CASE nState OF
    // Start by setting everything to a known value
    INIT:
        nState := WAIT_EXEC;
        bError := FALSE;
        sErrorMessage := '';
        bDone := FALSE;
        bCausedError := FALSE;
    // Normal "waiting for move command" state
    WAIT_EXEC:
        bMyMove := FALSE;
        // Looking for a rising edge on bExecute
        IF rtExec.Q THEN
            bDone := FALSE;
            nState := PICK_REQUEST;
        END_IF
    // Decide how to handle the request
    PICK_REQUEST:
        IF stMotionStage.bBusy THEN
            CASE enumMotionRequest OF
                ENUM_MotionRequest.WAIT:
                    nState := WAIT_OTHER_MOVE;
                ENUM_MotionRequest.INTERRUPT:
                    nState := STOP_OTHER_MOVE;
                ENUM_MotionRequest.ABORT:
                    nState := ERROR;
                    bError := TRUE;
                    nErrorId := 16#7900;
            END_CASE
        ELSE
            nState := START_MOVE;
        END_IF
    // Watch the other move, then see if it's our turn
    WAIT_OTHER_MOVE:
        IF NOT stMotionStage.bBusy THEN
            // Try to pick request again next cycle once the move is over
            nState := PICK_REQUEST;
        END_IF
    // Interrupt the other move, then go to start ours
    STOP_OTHER_MOVE:
        stMotionStage.bExecute := FALSE;
        IF NOT stMotionStage.bBusy THEN
            nState := START_MOVE;
        END_IF
    // Set the correct values on DUT_MotionStage to start a new absolute move
    START_MOVE:
        bMyMove := TRUE;
        stMotionStage.bExecute := TRUE;
        stMotionStage.nCommand := ENUM_EpicsMotorCmd.MOVE_ABSOLUTE;
        stMotionStage.fPosition := fPos;
        stMotionStage.fVelocity := fVel;
        stMotionStage.fAcceleration := fAcc;
        stMotionStage.fDeceleration := fDec;
        nState := WAIT_MY_MOVE;
    // Watch our ongoing move, look for the move to end or requests to stop the move from this FB
    WAIT_MY_MOVE:
        ftBusy(CLK:=stMotionStage.bBusy);
        IF ftBusy.Q THEN
            nState := DONE_MOVING;
        END_IF
        // Implement stop on falling trigger
        IF ftExec.Q THEN
            nState := STOP_MY_MOVE;
        END_IF
    // Request a stop and wait for it to happen
    STOP_MY_MOVE:
        stMotionStage.bExecute := FALSE;
        IF NOT stMotionStage.bBusy THEN
            nState := DONE_MOVING;
        END_IF
    // Pick out the bDone state and return to waiting
    DONE_MOVING:
        bDone := stMotionStage.bDone;
        nState := WAIT_EXEC;
    // Lock us into the error state until the FB is reset
    ERROR:
        bMyMove := FALSE;
END_CASE

// Transition to the ERROR state if applicable
IF bMyMove AND stMotionStage.bError THEN
    nState := ERROR;
    bError := TRUE;
    nErrorId := stMotionStage.nErrorId;
    bCausedError := TRUE;
END_IF
sErrorMessage := F_MotionErrorCodeLookup(nErrorId := nErrorId);

CASE nState OF
INIT, WAIT_EXEC, ERROR:
    bBusy := FALSE;
ELSE
    bBusy := TRUE;
END_CASE

END_FUNCTION_BLOCK

// POUs/Motion/States/FB_PositionStateLock
FUNCTION_BLOCK FB_PositionStateLock
(*
    Implements immutability for a locked DUT_PositionState
    Once this is called the first time, the parameters at the time of the call will be restored on all subsequent calls.
*)
VAR_IN_OUT
    stPositionState: DUT_PositionState;
END_VAR
VAR
    stCachedPositionState: DUT_PositionState;
    bInit: BOOL := FALSE;
END_VAR

// Force values to be cached if we've cached something
IF bInit AND stPositionState.bLocked THEN
    stPositionState.sName := stCachedPositionState.sName;
    stPositionState.fPosition := stCachedPositionState.fPosition;
    stPositionState.fDelta := stCachedPositionState.fDelta;
    stPositionState.fVelocity := stCachedPositionState.fVelocity;
    stPositionState.fAccel := stCachedPositionState.fAccel;
    stPositionState.fDecel := stCachedPositionState.fDecel;
// If we haven't cached and we should, make the cache. Note that we skip bLocked, bValid, and bMoveOk
ELSIF NOT bInit AND stPositionState.bLocked THEN
    stCachedPositionState.sName := stPositionState.sName;
    stCachedPositionState.fPosition := stPositionState.fPosition;
    stCachedPositionState.fDelta := stPositionState.fDelta;
    stCachedPositionState.fVelocity := stPositionState.fVelocity;
    stCachedPositionState.fAccel := stPositionState.fAccel;
    stCachedPositionState.fDecel := stPositionState.fDecel;
    bInit := TRUE;
// Do nothing, or unlock the state if bLocked goes FALSE
ELSIF NOT stPositionState.bLocked THEN
    bInit := FALSE;
END_IF

END_FUNCTION_BLOCK

// POUs/Motion/FB_MotionPneumaticActuator
(*This function blcok implements a pnuematic actuator. That can be signle or double acting by setting the ibSingleCntrl accordingly*)
(* with double acting ibCntrlHold signal should be false, while with single acting the signal should be true*)
FUNCTION_BLOCK FB_MotionPneumaticActuator
VAR_INPUT
    (*EPS Interlock Bits*)
    ibInsertOK: BOOL; (*Actuator can be Inserted*)
    ibRetractOK: BOOL; (*ACtuator can be retracted*)
    ibPMPS_OK:BOOL; (*to be linked the Arbiter bit*)
    ibSingleCntrl:BOOL;(* TRUE if Actuator requires one Output signal to be activated, FALSE if its double acting i.e two outputs are required*)
    ibCntrlHold:BOOL; (* Control Signal must retain its value, must be TRUE in the case of single acting*)
    ibOverrideInterlock:BOOL; (*if true interlocks are ignored*)
    // Reset fault
    {attribute 'pytmc' := '
    pv: FF_Reset
    '}
    i_xReset: BOOL;
END_VAR
VAR_OUTPUT
    {attribute 'pytmc' := '
    pv:
    '}
    stPneumaticActuator    :    DUT_MotionPneumaticActuator;
    {attribute 'pytmc' := '
     pv: MPS_OK
     field: ZNAM FALSE
     field: ONAM TRUE
     field: DESC TRUE if MPS signal is OK
    '}
    xMPS_OK:BOOL;
END_VAR
VAR_IN_OUT
    io_fbFFHWO    :    FB_HardwareFFOutput;
END_VAR
VAR
    // PMPS
    fbFF    :    FB_FastFault :=(
        i_DevName := 'MPA',
        i_Desc := 'Fault occurs when the device is moving',
        i_TypeCode := 10#1010);

    (*Init*)
    xFirstPass    :    BOOL;
    fbFSInit        :    R_TRIG;

    (* Timeouts*)
    tTimeOutDuration: TIME:= T#10S;
    tInserttimeout: TON;
    tRetracttimeout:TON;
    (*Limit switch latch timer*)
    tLimitSwitchLatchDuration: TIME:=T#1S;
    tInsertLimitSwitch:TON;
    tRetractLimitSwitch:TON;

    (*Logging*)
    fbLogger : FB_LogMessage := (eSubsystem:=E_SubSystem.MOTION);
    ePrevState : ENUM_PnuematicActuatorPositionState;
    tAction : R_TRIG; // Primary action of this device (Insert_DO, Retract_DO, etc.)
    tOverrideActivated : R_TRIG;

    (*IO*)
    i_xInsertedLS    AT%I*: BOOL;
    i_xRetractedLS    AT%I*: BOOL;
    q_xInsert_DO    AT%Q*: BOOL;
    q_xRetract_DO    AT%Q*: BOOL;

END_VAR


(*Initialize*)
fbFSInit( CLK := TRUE, Q => xFirstPass);
IF xFirstPass THEN
    stPneumaticActuator.eState := ENUM_PnuematicActuatorPositionState.INVALID;
    stPneumaticActuator.bRetract_SW := FALSE;
    stPneumaticActuator.bInsert_SW := FALSE;
END_IF

(*Soft IO Mapping to EPICS PVs*)
ACT_IO();

(* Manage States*)
IF stPneumaticActuator.i_bInLimitSwitch AND  stPneumaticActuator.i_bOutLimitSwitch THEN
    stPneumaticActuator.eState:=ENUM_PnuematicActuatorPositionState.INVALID;
ELSIF NOT stPneumaticActuator.i_bInLimitSwitch AND stPneumaticActuator.i_bOutLimitSwitch THEN
    stPneumaticActuator.eState:=ENUM_PnuematicActuatorPositionState.RETRACTED;
ELSIF stPneumaticActuator.i_bInLimitSwitch AND NOT stPneumaticActuator.i_bOutLimitSwitch THEN
    stPneumaticActuator.eState:=ENUM_PnuematicActuatorPositionState.INSERTED;
ELSIF NOT stPneumaticActuator.i_bInLimitSwitch AND NOT stPneumaticActuator.i_bOutLimitSwitch THEN
    stPneumaticActuator.eState:=ENUM_PnuematicActuatorPositionState.MOVING;
ELSE
    stPneumaticActuator.eState:=ENUM_PnuematicActuatorPositionState.INVALID ;
END_IF

(*Set the Done/Busy signal*)
stPneumaticActuator.bDone := (stPneumaticActuator.bRetract_SW AND stPneumaticActuator.eState=ENUM_PnuematicActuatorPositionState.RETRACTED)
                            OR (stPneumaticActuator.bInsert_SW AND stPneumaticActuator.eState=ENUM_PnuematicActuatorPositionState.INSERTED);
stPneumaticActuator.bBusy := (stPneumaticActuator.bRetract_SW AND stPneumaticActuator.eState<>ENUM_PnuematicActuatorPositionState.RETRACTED)
                            OR (stPneumaticActuator.bInsert_SW AND stPneumaticActuator.eState<>ENUM_PnuematicActuatorPositionState.INSERTED);
(*MPS FAULT*)
(* MPS Faults when the actuator is in motion*)
xMPS_OK := (stPneumaticActuator.eState=ENUM_PnuematicActuatorPositionState.RETRACTED) OR (stPneumaticActuator.eState=ENUM_PnuematicActuatorPositionState.INSERTED);
(*PMPS PERMISSION*)
// yet to be implemented

(* Can't have bRetract_SW and  bInsert_SW both be true*)
If (stPneumaticActuator.bRetract_SW) AND (stPneumaticActuator.bInsert_SW) THEN
    stPneumaticActuator.bRetract_SW := FALSE;
    stPneumaticActuator.bInsert_SW := FALSE;
END_IF
//Redundant??
(*Check if both digital outputs active at the same time, and clear all*)
IF stPneumaticActuator.q_bInsert THEN
    stPneumaticActuator.q_bRetract := FALSE;
    stPneumaticActuator.bRetract_SW:= FALSE;
END_IF;
IF stPneumaticActuator.q_bRetract THEN
    stPneumaticActuator.q_bInsert := FALSE;
    stPneumaticActuator.bInsert_SW:= FALSE;
END_IF;

(*Actuate the device*)
stPneumaticActuator.q_bRetract := stPneumaticActuator.bRetractOK AND stPneumaticActuator.bRetract_SW AND NOT stPneumaticActuator.bInsert_SW ;
stPneumaticActuator.q_bInsert := stPneumaticActuator.bInsertOK AND stPneumaticActuator.bInsert_SW AND NOT stPneumaticActuator.bRetract_SW ;

(*Reset the Control signal when command has been executed and give time to ensure the actuator is fully seated in either direction*)
IF (NOT ibSingleCntrl AND NOT ibCntrlHold) THEN
   IF (stPneumaticActuator.bRetract_SW AND stPneumaticActuator.i_bOutLimitSwitch AND tRetractLimitSwitch.Q ) THEN stPneumaticActuator.q_bRetract := FALSE; END_IF
   IF (stPneumaticActuator.bInsert_SW AND stPneumaticActuator.i_bInLimitSwitch AND tInsertLimitSwitch.Q) THEN stPneumaticActuator.q_bInsert := FALSE; END_IF
END_IF

(*Timers*)
tInserttimeout(IN:= stPneumaticActuator.q_bInsert, PT := tTimeOutDuration );
tRetracttimeout(IN:= stPneumaticActuator.q_bRetract, PT := tTimeOutDuration);
tInsertLimitSwitch(IN:= stPneumaticActuator.i_bInLimitSwitch, PT := tLimitSwitchLatchDuration);
tRetractLimitSwitch(IN:= stPneumaticActuator.i_bOutLimitSwitch, PT := tLimitSwitchLatchDuration);


///Check moving postion timout
IF NOT stPneumaticActuator.i_bInLimitSwitch AND tInserttimeout.Q THEN
    stPneumaticActuator.bError := TRUE;
    stPneumaticActuator.sErrorMessage:= 'Actuator insert timeout';
ELSIF NOT stPneumaticActuator.i_bOutLimitSwitch AND tRetracttimeout.Q THEN
    stPneumaticActuator.bError := TRUE;
    stPneumaticActuator.sErrorMessage:= 'Actuator retract timeout';
END_IF
// Reset error
stPneumaticActuator.bError R= stPneumaticActuator.bReset;

(*FAST FAULT*)
fbFF(i_xOK := xMPS_OK,
    i_xReset := i_xReset,
    io_fbFFHWO := io_fbFFHWO);

(*Soft IO Mapping to Epics pvs*)
ACT_IO();

ACTION ACT_IO:
(*Inputs*)
stPneumaticActuator.i_bInLimitSwitch :=  i_xInsertedLS;
stPneumaticActuator.i_bOutLimitSwitch := i_xRetractedLS;

(*outputs*)
q_xInsert_DO:=stPneumaticActuator.q_bInsert;
q_xRetract_DO:=stPneumaticActuator.q_bRetract;

(*EPICS*)
stPneumaticActuator.bRetractOK := ibRetractOK;
stPneumaticActuator.bInsertOK := ibInsertOK;
END_ACTION

ACTION ACT_Logger:
// Log Valve timeouts
IF (tInserttimeout.Q OR tRetracttimeout.Q) THEN fbLogger(sMsg:=stPneumaticActuator.sErrorMessage, eSevr:=TcEventSeverity.Warning); END_IF

// Log Actuator commands
// Log valve open
tAction(CLK:= (stPneumaticActuator.q_bRetract OR stPneumaticActuator.q_bInsert));
IF tAction.Q THEN
   IF(stPneumaticActuator.q_bRetract) THEN fbLogger(sMsg:='Actuator commanded retract', eSevr:=TcEventSeverity.Info); END_IF
   IF(stPneumaticActuator.q_bInsert) THEN fbLogger(sMsg:='Actuator commanded insert', eSevr:=TcEventSeverity.Info); END_IF
END_IF


// State Logging
IF ePrevState <> stPneumaticActuator.eState THEN
      CASE stPneumaticActuator.eState OF
        ENUM_PnuematicActuatorPositionState.INVALID:
            fbLogger(sMsg:='Actuator invalid position.', eSevr:=TcEventSeverity.Critical);
          ENUM_PnuematicActuatorPositionState.MOVING:
            fbLogger(sMsg:='Actuator moving', eSevr:=TcEventSeverity.Warning);
        ENUM_PnuematicActuatorPositionState.RETRACTED:
            fbLogger(sMsg:='Actuator Retracted.', eSevr:=TcEventSeverity.Info);
        ENUM_PnuematicActuatorPositionState.INSERTED:
            fbLogger(sMsg:='Actuator Inserted.', eSevr:=TcEventSeverity.Info);
      END_CASE
      ePrevState := stPneumaticActuator.eState;
  END_IF
END_ACTION

END_FUNCTION_BLOCK

// POUs/Motion/FB_MotionStageSim
FUNCTION_BLOCK FB_MotionStageSim
(*
    Set all the values needed for a fake motor to be movable
    via the IOC, then call FB_MotionStage
*)
VAR_IN_OUT
    stMotionStage: DUT_MotionStage;
END_VAR
VAR
    fbMotionStage: FB_MotionStage;
    bInit: BOOL;
END_VAR

IF NOT bInit THEN
    bInit := TRUE;
    // Stand-in for no forward limit
    stMotionStage.bLimitForwardEnable := TRUE;
    // Stand-in for no reverse limit
    stMotionStage.bLimitBackwardEnable := TRUE;
    // Stand-in for no STO button
    stMotionStage.bHardwareEnable := TRUE;
    // Stand-in for no PMPS governer
    stMotionStage.bPowerSelf := TRUE;
    // Always keep it enabled for testing ease
    stMotionStage.nEnableMode := ENUM_StageEnableMode.ALWAYS;
END_IF
// Call FB_MotionStage to do the thing
fbMotionStage(stMotionStage := stMotionStage);

END_FUNCTION_BLOCK

// POUs/MotorTesting/FB_MicroStepCountTest
FUNCTION_BLOCK FB_MicroStepCountTest
VAR_INPUT
    bExecute: BOOL;
    fStepSize: LREAL;
    nSteps: UINT;
    fMicroStep: LREAL;
    fVelocity: LREAL;
    tSettleTime: TIME;
END_VAR
VAR_IN_OUT
    Axis: AXIS_REF;
END_VAR
VAR_OUTPUT
    nStepsCounted: UINT;
    nTheorySteps: UINT;
    fPercent: LREAL;
    fEstMicroSize: LREAL;
END_VAR
VAR
    fbMoveRel: MC_MoveRelative;
    fbSettleTimer: TON;
    bDoMove: BOOL;
    nStepCounter: UINT;

    arrPosBuffer: ARRAY [0..99] OF LREAL;
    fAvgPos: LREAL;
    nArrIndex: UINT;
    nLoopIndex: UINT;

    fStartPos: LREAL;
    fPrevPos: LREAL;
    fStepChange: LREAL;

    fStepSum: LREAL;
END_VAR

// Motion FB
fbMoveRel(Axis:=Axis,
    Execute:=bDoMove,
    Distance:=fStepSize,
    Velocity:=fVelocity);

// Settle time
fbSettleTimer(IN:=fbMoveRel.Done,
    PT:=tSettleTime);

// Re-enable the move for next cycle
bDoMove := bExecute AND nStepCounter < nSteps;

// Calculate rolling average
arrPosBuffer[nArrIndex] := Axis.NcToPlc.ActPos;
fAvgPos := 0;
FOR nLoopIndex := 0 TO 99 DO
    fAvgPos := fAvgPos + arrPosBuffer[nLoopIndex];
END_FOR;
fAvgPos := fAvgPos / 100;
nArrIndex := (nArrIndex + 1) MOD 100;

// Initialize starting variables
IF NOT bExecute THEN
    fStartPos := fAvgPos;
    fPrevPos := fAvgPos;
END_IF

// Check results
IF fbSettleTimer.Q THEN
    fStepChange := fAvgPos - fPrevPos;
    // Invert fStepChange if we were doing negative steps
    IF fStepSize < 0 THEN
        fStepChange := fStepChange * -1;
    END_IF
    IF fStepChange > fMicroStep * 0.5 THEN
        nStepsCounted := nStepsCounted + 1;
        fStepSum := fStepSum + fStepChange;
        fEstMicroSize := fStepSum / nStepsCounted;
    END_IF
    nTheorySteps := DINT_TO_UINT(TRUNC(ABS((fStartPos - fAvgPos) / fMicroStep)));
    IF nTheorySteps > 0 THEN
        fPercent := 100 * nStepsCounted / nTheorySteps;
    END_IF
    fPrevPos := fAvgPos;
    nStepCounter := nStepCounter + 1;
    // Reset the move block
    bDoMove := FALSE;
END_IF

END_FUNCTION_BLOCK

// tc_mca_std_lib/POUs/ErrorHandling/FB_ErrorList
FUNCTION_BLOCK FB_ErrorList

VAR_INPUT
	En : BOOL;											//Enable input
	bReset : BOOL;										//Delete all Error entry
	lErrorID : ULINT;									//ErrorID to be acknoledged
	bACK : BOOL;										//Acknoledge the given error and delete it from the list
END_VAR
	
VAR_OUTPUT
	EnO : BOOL;											//Enable output
	nNoError: UINT;										//Number of Errors
	nNoOverflow : INT;									//Number of Overflows
	pErrorSystem : POINTER TO ST_ErrorSystem;			//Pointer to ErrorSystem
END_VAR

VAR
	nFreePos : UINT;									//Number of free position in the list
	nListCnt1 : UINT;									//work variable
	ErrorSystem : ST_ErrorSystem;						//Data structure of the Error list
END_VAR

(*
* ================================================================================
*                                   DESCRIPTION
* ================================================================================
* This Function Block implements the core structure of the Error/Warning Handling
* system. It realizes the datastructure containing every Error Entry, collect
* statistics about the usage and manage the Error Entries.
* Note: The system is under development, most of the functionalities are not
* implemented or existing functionalities may change with time.
* ================================================================================
*)
EnO := En;

//Ponter to ErrorSystem
pErrorSystem := ADR(ErrorSystem);

//Number of overflows
nNoOverflow := ErrorSystem.nNoOverflows;

IF bReset THEN
	MEMSET ( ADR(ErrorSystem.aErrorData[0]), 0, GVL_ErrorSystem.cSizeOfErrorData * SIZEOF(DUT_TerminalError));
	ErrorSystem.lNextErrorID := 1;
END_IF

//Number of errors in the system
nNoError := 0;
FOR nListCnt1 := 0 TO GVL_ErrorSystem.cSizeOfErrorData - 1 DO
	IF ErrorSystem.aErrorData[nListCnt1].Error_ID <> 0  THEN
		nNoError := nNoError+1; 
	END_IF
END_FOR
ErrorSystem.nNoErrors := nNoError;

//Number of free position in the list
nFreePos := GVL_ErrorSystem.cSizeOfErrorData - nNoError;

//Acknoledge specified Error entry
IF bACK THEN
	FOR nListCnt1 := 0 TO GVL_ErrorSystem.cSizeOfErrorData - 1 DO
		IF ErrorSystem.aErrorData[nListCnt1].Error_ID = lErrorID THEN
			ErrorSystem.aErrorData[nListCnt1].ErrorState := DUT_ErrorState.Acknowledged;
		END_IF
	END_FOR
END_IF

//Deleting acknoledged errors
FOR nListCnt1 := 0 TO GVL_ErrorSystem.cSizeOfErrorData - 1 DO
	IF ErrorSystem.aErrorData[nListCnt1].ErrorState = DUT_ErrorState.Acknowledged THEN
		MEMMOVE (ADR(ErrorSystem.aErrorData[nListCnt1]), ADR(ErrorSystem.aErrorData[nListCnt1+1]), (GVL_ErrorSystem.cSizeOfErrorData - 1 - nListCnt1) * SIZEOF(DUT_TerminalError));
		MEMSET(ADR(ErrorSystem.aErrorData[GVL_ErrorSystem.cSizeOfErrorData - 1]), 0, SIZEOF(DUT_TerminalError));
	END_IF
END_FOR

END_FUNCTION_BLOCK

// tc_mca_std_lib/POUs/ErrorHandling/FB_TerminalError
FUNCTION_BLOCK FB_TerminalError

VAR_INPUT
	En					: BOOL;
	iTerminal_ID		: INT;
	bWcState			: BOOL;
	uiInfoData_State	: UINT;
	pErrorSystem		: POINTER TO ST_ErrorSystem;					//Pointer to the error system
END_VAR

VAR_OUTPUT
	EnO : BOOL;
	bError : BOOL := FALSE;
END_VAR

VAR
	iStateError : UINT;
	iOtherError : UINT;
	ErrorData	: DUT_TerminalError;
	nErrSysCNT	: UINT;
	
	//testing
	bStateChanged : BOOL;						//Indicate if state change happened
	uiInfoData_State_Prev : UINT := 16#8;		//Previous value of Infodata.State
	bWcState_Prev : BOOL := FALSE;				//Previous state of WcState
	
	//FB-s
	
END_VAR

(*
Currently:

Problem:

TODO:

*)

//Connect EN to EnO
EnO:=En;

//Check if pointer is OK
IF pErrorSystem=0 THEN RETURN; END_IF

//Any difference from normal state creates an error
IF En AND (bWcState OR uiInfoData_State<>16#8) THEN
	bError:=TRUE;
ELSE
	bError:=FALSE;
END_IF

//Change detection
IF uiInfoData_State <> uiInfoData_State_Prev OR bWcState <> bWcState_Prev THEN
	bStateChanged := TRUE;
ELSE
	bStateChanged := FALSE;
END_IF

//Update previous values
uiInfoData_State_Prev := uiInfoData_State;
bWcState_Prev := bWcState;

//Decision tree
IF bStateChanged THEN
	IF bError THEN
		IF ErrorData.ErrorState = DUT_ErrorState.Active THEN
			//Close active error
			//Read system time
			ErrorData.nDateTimeOff := Tc2_EtherCAT.F_GetActualDcTime64();
			ErrorData.sDateTimeOff := Tc2_EtherCat.DCTIME64_TO_STRING(ErrorData.nDateTimeOff);
			ErrorData.ErrorState := DUT_ErrorState.Inactive;
			//Write Off-time to Error System
			FOR nErrSysCNT := 0 TO GVL_ErrorSystem.cSizeOfErrorData - 1 DO
				IF pErrorSystem^.aErrorData[nErrSysCNT].Error_ID = ErrorData.Error_ID THEN
					pErrorSystem^.aErrorData[nErrSysCNT].nDateTimeOff := ErrorData.nDateTimeOff;
					pErrorSystem^.aErrorData[nErrSysCNT].sDateTimeOff := ErrorData.sDateTimeOff;
					pErrorSystem^.aErrorData[nErrSysCNT].ErrorState := DUT_ErrorState.Inactive;
					EXIT;
				END_IF
			END_FOR
				
			//Clear ErrorData
			MEMSET(ADR(ErrorData), 0, SIZEOF(ErrorData));
		END_IF
		
		//Open a new error
		ErrorData.ErrorState := DUT_ErrorState.Active;												//Set Error State
		ErrorData.nDateTimeOn := Tc2_EtherCAT.F_GetActualDcTime64();								//Get system time
		ErrorData.sDateTimeOn := Tc2_EtherCat.DCTIME64_TO_STRING(ErrorData.nDateTimeOn);			//Convert to string
		ErrorData.iTerminalID := iTerminal_ID;														//Terminal_ID
		ErrorData.bWcState := bWcState;																//WcState bit
		ErrorData.uiInfoDataState := uiInfoData_State;												//uiInfoData_State
		
		//Error message according to uiInfoData_State and WcState
		iStateError := (uiInfoData_State AND 16#000F);												//Mask for operation state 
		iOtherError := (uiInfoData_State AND 16#00F0);												//Mask for the other 3 kind of errors
		//Error messages according to the least significant digit
		CASE iStateError OF
			16#0001 : ErrorData.sErrorMessage := 'Slave in INIT state;   ';
			16#0002 : ErrorData.sErrorMessage := 'Slave in PREOP state;   ';
			16#0003 : ErrorData.sErrorMessage := 'Slave in BOOT state;   ';
			16#0004 : ErrorData.sErrorMessage := 'Slave in SAFEOP state;   ';
			16#0008 : ;																			//Normal operation state
		ELSE
			ErrorData.sErrorMessage := 'Undefined State of operation;   ';						//I hope we will never see this message
			ErrorData.sErrorMessage := CONCAT (ErrorData.sErrorMessage, UINT_TO_STRING(iStateError));
			ErrorData.sErrorMessage := CONCAT (ErrorData.sErrorMessage, '   ');
		END_CASE
		
		//Error messages according to the second least significant digit
		CASE iOtherError OF
			16#0000 : ;																			//No error case
			16#0010 : ErrorData.sErrorMessage := CONCAT (ErrorData.sErrorMessage, 'Slave signals error;   ');
			16#0020 : ErrorData.sErrorMessage := CONCAT (ErrorData.sErrorMessage, 'Invalid vendorID/productCode read;   ');
			16#0040 : ErrorData.sErrorMessage := CONCAT (ErrorData.sErrorMessage, 'Initialisation error occured;   ');
		ELSE
			ErrorData.sErrorMessage := CONCAT (ErrorData.sErrorMessage, 'Undefined Error ID: ');
			ErrorData.sErrorMessage := CONCAT (ErrorData.sErrorMessage, UINT_TO_STRING(iOtherError));
			ErrorData.sErrorMessage := CONCAT (ErrorData.sErrorMessage, '   ');
		END_CASE
	
		//Errormessage according to WcState bit
		IF bWcState THEN
			ErrorData.sErrorMessage := CONCAT (ErrorData.sErrorMessage, 'Invalid Data;');
		END_IF
		
		//Check for overflow
		IF pErrorSystem^.nNoErrors = GVL_ErrorSystem.cSizeOfErrorData THEN
			pErrorSystem^.nNoOverflows := pErrorSystem^.nNoOverflows+1;
		END_IF
		
		//Write Error Data into Error System
		ErrorData.Error_ID := pErrorSystem^.lNextErrorID ;
		MEMMOVE( ADR(pErrorSystem^.aErrorData[1]), ADR(pErrorSystem^.aErrorData[0]), (GVL_ErrorSystem.cSizeOfErrorData-1) * SIZEOF(DUT_TerminalError));
		pErrorSystem^.aErrorData[0] := ErrorData;
		pErrorSystem^.lNextErrorID := pErrorSystem^.lNextErrorID+1;
		
	ELSE
		//Close Active Error
		//Read system time
		ErrorData.nDateTimeOff := Tc2_EtherCAT.F_GetActualDcTime64();
		ErrorData.sDateTimeOff := Tc2_EtherCat.DCTIME64_TO_STRING(ErrorData.nDateTimeOff);
		ErrorData.ErrorState := DUT_ErrorState.Inactive;
		
		//Write Off time to Error System
		FOR nErrSysCNT := 0 TO GVL_ErrorSystem.cSizeOfErrorData - 1 DO
			IF pErrorSystem^.aErrorData[nErrSysCNT].Error_ID = ErrorData.Error_ID THEN
				pErrorSystem^.aErrorData[nErrSysCNT].nDateTimeOff := ErrorData.nDateTimeOff;
				pErrorSystem^.aErrorData[nErrSysCNT].sDateTimeOff := ErrorData.sDateTimeOff;
				pErrorSystem^.aErrorData[nErrSysCNT].ErrorState := DUT_ErrorState.Inactive;
				EXIT;
			END_IF
		END_FOR
			
		//Clear ErrorData
		MEMSET(ADR(ErrorData), 0, SIZEOF(ErrorData));
	END_IF
END_IF

END_FUNCTION_BLOCK

// tc_mca_std_lib/POUs/Hardware/EtherCAT_Terminals/Analog_Inputs/EL3174_0002
//EL3174-0002 | 4-channel analog input, -10/0...+10V, -20/0/+4...20mA, 16 bit, differential
FUNCTION_BLOCK EL3174_0002

VAR_INPUT
	En: BOOL;
	iTerminal_ID : INT;
	ErrorSystem : POINTER TO ST_ErrorSystem;
END_VAR
	
VAR_OUTPUT
	EnO: BOOL;
	iAi_Ch1_Value : INT;
	iAi_Ch2_Value : INT;
	iAi_Ch3_Value : INT;
	iAi_Ch4_Value : INT;
	bError: BOOL;
END_VAR

VAR
	//Channels
	AI_Std_Ch_1_Status	AT %I* : WORD;
	AI_Std_Ch_1_Value 	AT %I* : INT;
	AI_Std_Ch_2_Status 	AT %I* : WORD;
	AI_Std_Ch_2_Value 	AT %I* : INT;
	AI_Std_Ch_3_Status 	AT %I* : WORD;
	AI_Std_Ch_3_Value 	AT %I* : INT;
	AI_Std_Ch_4_Status 	AT %I* : WORD;
	AI_Std_Ch_4_Value 	AT %I* : INT;
	
	//Terminal status
	WcState_WcState AT %I*: BOOL;
	InfoData_State AT %I*: UINT;
	
	//FB-s
	EL3174_0002_Error : FB_TerminalError;
END_VAR

(*
* TODO:
* Status words of the channels
*)

EnO := En;

//Error FB instance
EL3174_0002_Error(
	En := TRUE,
	iTerminal_ID := iTerminal_ID,
	bWcState := WcState_WcState,
	uiInfoData_State := InfoData_State,
	pErrorSystem := ErrorSystem,
	bError => bError,
);

IF En THEN
	IF bError = FALSE THEN
		iAi_Ch1_Value := AI_Std_Ch_1_Value;
		iAi_Ch2_Value := AI_Std_Ch_2_Value;
		iAi_Ch3_Value := AI_Std_Ch_3_Value;
		iAi_Ch4_Value := AI_Std_Ch_4_Value;
	ELSE
		iAi_Ch1_Value := 0;
		iAi_Ch2_Value := 0;
		iAi_Ch3_Value := 0;
		iAi_Ch4_Value := 0;
	END_IF
END_IF

END_FUNCTION_BLOCK

// tc_mca_std_lib/POUs/Hardware/EtherCAT_Terminals/Analog_Inputs/EL3214
//EL3214 | 4-channel analog input terminal, PT100 (RTD)
FUNCTION_BLOCK EL3214

VAR_INPUT
	En: BOOL;
	iTerminal_ID : INT;
	ErrorSystem : POINTER TO ST_ErrorSystem;
END_VAR

VAR_OUTPUT
	EnO: BOOL;
	iAi_Ch1_Value : INT;
	iAi_Ch2_Value : INT;
	iAi_Ch3_Value : INT;
	iAi_Ch4_Value : INT;
	bError: BOOL;
END_VAR

VAR
	//Channels
	AI_RTD_Ch_1_Status	AT %I* : WORD;
	AI_RTD_Ch_1_Value 	AT %I* : INT;
	AI_RTD_Ch_2_Status 	AT %I* : WORD;
	AI_RTD_Ch_2_Value 	AT %I* : INT;
	AI_RTD_Ch_3_Status 	AT %I* : WORD;
	AI_RTD_Ch_3_Value 	AT %I* : INT;
	AI_RTD_Ch_4_Status 	AT %I* : WORD;
	AI_RTD_Ch_4_Value 	AT %I* : INT;
	
	//Terminal status
	WcState_WcState AT %I*: BOOL;
	InfoData_State AT %I*: UINT;
	
	//FB-s
	EL3214_Error : FB_TerminalError;
END_VAR

(*
* TODO:
* Status words of the channels
*)

EnO := En;

//Error FB instance
EL3214_Error(
	En := TRUE,
	iTerminal_ID := iTerminal_ID,
	bWcState := WcState_WcState,
	uiInfoData_State := InfoData_State,
	pErrorSystem := ErrorSystem,
	bError => bError,
);

IF En THEN
	IF bError = FALSE THEN
		iAi_Ch1_Value := AI_RTD_Ch_1_Value;
		iAi_Ch2_Value := AI_RTD_Ch_2_Value;
		iAi_Ch3_Value := AI_RTD_Ch_3_Value;
		iAi_Ch4_Value := AI_RTD_Ch_4_Value;
	ELSE
		iAi_Ch1_Value := 0;
		iAi_Ch2_Value := 0;
		iAi_Ch3_Value := 0;
		iAi_Ch4_Value := 0;
	END_IF
END_IF

END_FUNCTION_BLOCK

// tc_mca_std_lib/POUs/Hardware/EtherCAT_Terminals/Analog_Inputs/EL3255
//EL3255 | 5-channel potentiometer measurement with sensor supply
FUNCTION_BLOCK EL3255

VAR_INPUT
	En: BOOL;
	iTerminal_ID : INT;
	ErrorSystem : POINTER TO ST_ErrorSystem;
END_VAR

VAR_OUTPUT
	EnO : BOOL;	
	Ch1_Value : INT;
	Ch2_Value : INT;
	Ch3_Value : INT;
	Ch4_Value : INT;
	Ch5_Value : INT;
	bError : BOOL;
END_VAR

VAR
	AI_Std_Ch1_Value AT %I* : INT;
	AI_Std_Ch2_Value AT %I* : INT;
	AI_Std_Ch3_Value AT %I* : INT;
	AI_Std_Ch4_Value AT %I* : INT;
	AI_Std_Ch5_Value AT %I* : INT;
	WcState_WcState AT %I*: BOOL;
	InfoData_State AT %I*: UINT;
	
	//FB-s
	EL3255_Error : FB_TerminalError;
END_VAR

(*
* TODO:
* Channel Status words
*)

EnO:=En;

//Error FB instance
EL3255_Error(
	En := TRUE,
	iTerminal_ID := iTerminal_ID,
	bWcState := WcState_WcState,
	uiInfoData_State := InfoData_State,
	pErrorSystem := ErrorSystem,
	bError => bError,
);

IF EN THEN
	IF NOT bError THEN
		Ch1_Value := AI_Std_Ch1_Value;
		Ch2_Value := AI_Std_Ch2_Value;
		Ch3_Value := AI_Std_Ch3_Value;
		Ch4_Value := AI_Std_Ch4_Value;
		Ch5_Value := AI_Std_Ch5_Value;
	ELSE
		Ch1_Value := 0;
		Ch2_Value := 0;
		Ch3_Value := 0;
		Ch4_Value := 0;
		Ch5_Value := 0;
	END_IF
END_IF

END_FUNCTION_BLOCK

// tc_mca_std_lib/POUs/Hardware/EtherCAT_Terminals/Analog_Inputs/FB_CalculateFrequency_3702_v0_01
FUNCTION_BLOCK FB_CalculateFrequency_3702_v0_01
VAR CONSTANT
	///200 samples/period
	cBufferSize: INT := 1000;
END_VAR
VAR_INPUT
	En: BOOL;
	bCalculate: BOOL;
	aBufferValue: ARRAY[0..(cBuffersize - 1)] OF INT;
	aBufferDcTime: ARRAY[0..(cBuffersize - 1)] OF UDINT;
	///If curve has a DC offset
	nDCOffset: INT := 0;
END_VAR
VAR_OUTPUT
	EnO: BOOL;
	bError: BOOL;
	fActFrequency: LREAL;
END_VAR
VAR
	nIndex: INT;
	nFirstZeroCrossing: INT;
	nLastZeroCrossing: INT;
	rTimeFirst: REAL := 0;
	rTimeLast: REAL := 0;
	rTimeRes: REAL := 0;
	nCrossings: INT := 0;
END_VAR
VAR_TEMP
	rRange: REAL := 0;
	rTimeSpan: REAL := 0;
END_VAR

EnO:=En;
bError:=FALSE;
nCrossings:=0;
IF En AND bCalculate THEN
	//Serach for crossings of nDCOffset
	FOR nIndex:=1 TO cBuffersize-1 DO
		IF((aBufferValue[nIndex]>nDCOffset AND aBufferValue[nIndex-1]<=nDCOffset) OR (aBufferValue[nIndex]<nDCOffset AND aBufferValue[nIndex-1]>=nDCOffset))	THEN
			IF(nCrossings=0) THEN
				nFirstZeroCrossing:=nIndex;
			END_IF
			nLastZeroCrossing:=nIndex;
			nCrossings:=nCrossings+1;
		END_IF
	END_FOR	
	
	IF nFirstZeroCrossing < nLastZeroCrossing  AND  nCrossings>2 THEN
		//interpolate zero crossings for higher accuracy
		rTimeRes:=UDINT_TO_REAL(aBufferDcTime[1]-aBufferDcTime[0]); //Buffer must contain more than 2 values
		rRange:=INT_TO_REAL(ABS(aBufferValue[nFirstZeroCrossing-1]-aBufferValue[nFirstZeroCrossing]));
		rTimeFirst:=UDINT_TO_REAL( aBufferDcTime[nFirstZeroCrossing-1])+ABS(INT_TO_REAL(aBufferValue[nFirstZeroCrossing-1])/rRange*rTimeRes);
		rRange:=INT_TO_REAL(ABS(aBufferValue[nLastZeroCrossing-1]-aBufferValue[nLastZeroCrossing]));
		rTimeLast:=UDINT_TO_REAL( aBufferDcTime[nLastZeroCrossing-1])+ABS(INT_TO_REAL(aBufferValue[nLastZeroCrossing-1])/rRange*rTimeRes);

		//Time span first to last (considering that max one time counter overflow have occured in the total time range of the time buffer)	
		IF rTimeFirst<rTimeLast THEN		
			rTimeSpan:=rTimeLast-rTimeFirst;
		ELSE //overflow of counter once (only 32bit timestamp =4.29seconds)
			rTimeSpan:=4294967296.0-rTimeFirst+rTimeLast;
		END_IF
		
		fActFrequency:=1000000000.0/rTimeSpan*(nCrossings-1)/2; //two crossings per period => Average frequency over buffer.
	ELSE
		fActFrequency:=0;
	END_IF
END_IF

END_FUNCTION_BLOCK

// tc_mca_std_lib/POUs/Hardware/EtherCAT_Terminals/Digital_Inputs/EL1008
///EL1008 | 8-channel digital input terminal 24 V DC, 3 ms
FUNCTION_BLOCK EL1008

VAR_INPUT
	En: BOOL;
	iTerminal_ID : INT;
	ErrorSystem : POINTER TO ST_ErrorSystem;
END_VAR

VAR_OUTPUT
	EnO: BOOL;
	bDi_1: BOOL;
	bDi_2: BOOL;
	bDi_3: BOOL;
	bDi_4: BOOL;
	bDi_5: BOOL;
	bDi_6: BOOL;
	bDi_7: BOOL;
	bDi_8: BOOL;
	bError: BOOL;
END_VAR

VAR
	Channel_1_Input AT %I*: BOOL;
	Channel_2_Input AT %I*: BOOL;
	Channel_3_Input AT %I*: BOOL;
	Channel_4_Input AT %I*: BOOL;
	Channel_5_Input AT %I*: BOOL;
	Channel_6_Input AT %I*: BOOL;
	Channel_7_Input AT %I*: BOOL;
	Channel_8_Input AT %I*: BOOL;
	WcState_WcState AT %I*: BOOL;
	InfoData_State AT %I*: UINT;
	
	//FB-s
	EL1008_Error : FB_TerminalError;
END_VAR

EnO:=En;

//Error FB instance
EL1008_Error(
	En := TRUE,
	iTerminal_ID := iTerminal_ID,
	bWcState := WcState_WcState,
	uiInfoData_State := InfoData_State,
	pErrorSystem := ErrorSystem,
	bError => bError,
);

IF En THEN
	IF bError=FALSE THEN
		bDi_1:=Channel_1_Input;
		bDi_2:=Channel_2_Input;
		bDi_3:=Channel_3_Input;
		bDi_4:=Channel_4_Input;
		bDi_5:=Channel_5_Input;
		bDi_6:=Channel_6_Input;
		bDi_7:=Channel_7_Input;
		bDi_8:=Channel_8_Input;
	ELSE
		bDi_1:=FALSE;
		bDi_2:=FALSE;
		bDi_3:=FALSE;
		bDi_4:=FALSE;
		bDi_5:=FALSE;
		bDi_6:=FALSE;
		bDi_7:=FALSE;
		bDi_8:=FALSE;
	END_IF
END_IF

END_FUNCTION_BLOCK

// tc_mca_std_lib/POUs/Hardware/EtherCAT_Terminals/Digital_Inputs/EL1018
///EL1018 | 8-channel digital input terminal 24 V DC, 10 µs
FUNCTION_BLOCK EL1018

VAR_INPUT
	En: BOOL;
	iTerminal_ID : INT;
	ErrorSystem : POINTER TO ST_ErrorSystem;
END_VAR

VAR_OUTPUT
	EnO: BOOL;
	bDi_1: BOOL;
	bDi_2: BOOL;
	bDi_3: BOOL;
	bDi_4: BOOL;
	bDi_5: BOOL;
	bDi_6: BOOL;
	bDi_7: BOOL;
	bDi_8: BOOL;
	bError : BOOL;
END_VAR

VAR
	Channel_1_Input AT %I*: BOOL;
	Channel_2_Input AT %I*: BOOL;
	Channel_3_Input AT %I*: BOOL;
	Channel_4_Input AT %I*: BOOL;
	Channel_5_Input AT %I*: BOOL;
	Channel_6_Input AT %I*: BOOL;
	Channel_7_Input AT %I*: BOOL;
	Channel_8_Input AT %I*: BOOL;
	WcState_WcState AT %I*: BOOL;
	InfoData_State  AT %I*: UINT;
	
	//FB-s
	EL1018_Error : FB_TerminalError;
END_VAR

EnO:=En;

//Error FB instance
EL1018_Error(
	En := TRUE,
	iTerminal_ID := iTerminal_ID,
	bWcState := WcState_WcState,
	uiInfoData_State := InfoData_State,
	pErrorSystem := ErrorSystem,
	bError => bError,
);

IF En THEN
	IF bError=FALSE THEN
		bDi_1:=Channel_1_Input;
		bDi_2:=Channel_2_Input;
		bDi_3:=Channel_3_Input;
		bDi_4:=Channel_4_Input;
		bDi_5:=Channel_5_Input;
		bDi_6:=Channel_6_Input;
		bDi_7:=Channel_7_Input;
		bDi_8:=Channel_8_Input;
	ELSE
		bDi_1:=FALSE;
		bDi_2:=FALSE;
		bDi_3:=FALSE;
		bDi_4:=FALSE;
		bDi_5:=FALSE;
		bDi_6:=FALSE;
		bDi_7:=FALSE;
		bDi_8:=FALSE;
	END_IF
END_IF

END_FUNCTION_BLOCK

// tc_mca_std_lib/POUs/Hardware/EtherCAT_Terminals/Digital_Inputs/EL1808
///EL1808 | HD EtherCAT Terminals, 8-channel digital input 24 V DC, 3 ms, 2-wire connection
FUNCTION_BLOCK EL1808

VAR_INPUT
	En: BOOL;
	iTerminal_ID : INT;
	ErrorSystem : POINTER TO ST_ErrorSystem;
END_VAR

VAR_OUTPUT
	EnO: BOOL;
	bDi_1: BOOL;
	bDi_2: BOOL;
	bDi_3: BOOL;
	bDi_4: BOOL;
	bDi_5: BOOL;
	bDi_6: BOOL;
	bDi_7: BOOL;
	bDi_8: BOOL;
	bError: BOOL;
END_VAR

VAR
	Channel_1_Input AT %I*: BOOL;
	Channel_2_Input AT %I*: BOOL;
	Channel_3_Input AT %I*: BOOL;
	Channel_4_Input AT %I*: BOOL;
	Channel_5_Input AT %I*: BOOL;
	Channel_6_Input AT %I*: BOOL;
	Channel_7_Input AT %I*: BOOL;
	Channel_8_Input AT %I*: BOOL;
	WcState_WcState AT %I*: BOOL;
	InfoData_State AT %I*: UINT;
	
	//FB-s
	EL1808_Error : FB_TerminalError;
END_VAR

EnO:=En;

//Error FB instance
EL1808_Error(
	En := TRUE,
	iTerminal_ID := iTerminal_ID,
	bWcState := WcState_WcState,
	uiInfoData_State := InfoData_State,
	pErrorSystem := ErrorSystem,
	bError => bError,
);

IF En THEN
	IF bError=FALSE THEN
		bDi_1:=Channel_1_Input;
		bDi_2:=Channel_2_Input;
		bDi_3:=Channel_3_Input;
		bDi_4:=Channel_4_Input;
		bDi_5:=Channel_5_Input;
		bDi_6:=Channel_6_Input;
		bDi_7:=Channel_7_Input;
		bDi_8:=Channel_8_Input;
	ELSE
		bDi_1:=FALSE;
		bDi_2:=FALSE;
		bDi_3:=FALSE;
		bDi_4:=FALSE;
		bDi_5:=FALSE;
		bDi_6:=FALSE;
		bDi_7:=FALSE;
		bDi_8:=FALSE;
	END_IF
END_IF

END_FUNCTION_BLOCK

// tc_mca_std_lib/POUs/Hardware/EtherCAT_Terminals/Digital_Inputs/EL1809
///EL1809 | HD EtherCAT Terminals, 16-channel digital input 24 V DC, 3 ms
FUNCTION_BLOCK EL1809

VAR_INPUT
	En: BOOL;
	iTerminal_ID : INT;
	ErrorSystem : POINTER TO ST_ErrorSystem;
END_VAR

VAR_OUTPUT
	EnO: BOOL;
	bDi_1: BOOL;
	bDi_2: BOOL;
	bDi_3: BOOL;
	bDi_4: BOOL;
	bDi_5: BOOL;
	bDi_6: BOOL;
	bDi_7: BOOL;
	bDi_8: BOOL;
	bDi_9: BOOL;
	bDi_10: BOOL;
	bDi_11: BOOL;
	bDi_12: BOOL;
	bDi_13: BOOL;
	bDi_14: BOOL;
	bDi_15: BOOL;
	bDi_16: BOOL;
	bError: BOOL;
END_VAR

VAR
	Channel_1_Input AT %I*: BOOL;
	Channel_2_Input AT %I*: BOOL;
	Channel_3_Input AT %I*: BOOL;
	Channel_4_Input AT %I*: BOOL;
	Channel_5_Input AT %I*: BOOL;
	Channel_6_Input AT %I*: BOOL;
	Channel_7_Input AT %I*: BOOL;
	Channel_8_Input AT %I*: BOOL;
	Channel_9_Input AT %I*: BOOL;
	Channel_10_Input AT %I*: BOOL;
	Channel_11_Input AT %I*: BOOL;
	Channel_12_Input AT %I*: BOOL;
	Channel_13_Input AT %I*: BOOL;
	Channel_14_Input AT %I*: BOOL;
	Channel_15_Input AT %I*: BOOL;
	Channel_16_Input AT %I*: BOOL;
	WcState_WcState AT %I*: BOOL;
	InfoData_State AT %I*: UINT;
	
	//FB-s
	EL1809_Error : FB_TerminalError;
END_VAR

EnO:=En;

//Error FB instance
EL1809_Error(
	En := TRUE,
	iTerminal_ID := iTerminal_ID,
	bWcState := WcState_WcState,
	uiInfoData_State := InfoData_State,
	pErrorSystem := ErrorSystem,
	bError => bError,
);

IF En THEN
	IF bError=FALSE THEN
		bDi_1:=Channel_1_Input;
		bDi_2:=Channel_2_Input;
		bDi_3:=Channel_3_Input;
		bDi_4:=Channel_4_Input;
		bDi_5:=Channel_5_Input;
		bDi_6:=Channel_6_Input;
		bDi_7:=Channel_7_Input;
		bDi_8:=Channel_8_Input;
		bDi_9:=Channel_9_Input;
		bDi_10:=Channel_10_Input;
		bDi_11:=Channel_11_Input;
		bDi_12:=Channel_12_Input;
		bDi_13:=Channel_13_Input;
		bDi_14:=Channel_14_Input;
		bDi_15:=Channel_15_Input;
		bDi_16:=Channel_16_Input;
	ELSE
		bDi_1:=FALSE;
		bDi_2:=FALSE;
		bDi_3:=FALSE;
		bDi_4:=FALSE;
		bDi_5:=FALSE;
		bDi_6:=FALSE;
		bDi_7:=FALSE;
		bDi_8:=FALSE;
		bDi_9:=FALSE;
		bDi_10:=FALSE;
		bDi_11:=FALSE;
		bDi_12:=FALSE;
		bDi_13:=FALSE;
		bDi_14:=FALSE;
		bDi_15:=FALSE;
		bDi_16:=FALSE;
	END_IF
END_IF

END_FUNCTION_BLOCK

// tc_mca_std_lib/POUs/Hardware/EtherCAT_Terminals/Digital_Inputs/EL1819
///EL1819 | HD EtherCAT Terminals, 16-channel digital input 24 V DC, 10 µs
FUNCTION_BLOCK EL1819

VAR_INPUT
	En: BOOL;
	iTerminal_ID : INT;
	ErrorSystem : POINTER TO ST_ErrorSystem;
END_VAR

VAR_OUTPUT
	EnO: BOOL;
	bDi_1: BOOL;
	bDi_2: BOOL;
	bDi_3: BOOL;
	bDi_4: BOOL;
	bDi_5: BOOL;
	bDi_6: BOOL;
	bDi_7: BOOL;
	bDi_8: BOOL;
	bDi_9: BOOL;
	bDi_10: BOOL;
	bDi_11: BOOL;
	bDi_12: BOOL;
	bDi_13: BOOL;
	bDi_14: BOOL;
	bDi_15: BOOL;
	bDi_16: BOOL;
	bError: BOOL;
END_VAR

VAR
	Channel_1_Input AT %I*: BOOL;
	Channel_2_Input AT %I*: BOOL;
	Channel_3_Input AT %I*: BOOL;
	Channel_4_Input AT %I*: BOOL;
	Channel_5_Input AT %I*: BOOL;
	Channel_6_Input AT %I*: BOOL;
	Channel_7_Input AT %I*: BOOL;
	Channel_8_Input AT %I*: BOOL;
	Channel_9_Input AT %I*: BOOL;
	Channel_10_Input AT %I*: BOOL;
	Channel_11_Input AT %I*: BOOL;
	Channel_12_Input AT %I*: BOOL;
	Channel_13_Input AT %I*: BOOL;
	Channel_14_Input AT %I*: BOOL;
	Channel_15_Input AT %I*: BOOL;
	Channel_16_Input AT %I*: BOOL;
	WcState_WcState AT %I*: BOOL;
	InfoData_State AT %I*: UINT;
	
	//FB-s
	EL1819_Error : FB_TerminalError;
END_VAR

EnO:=En;

//Error FB instance
EL1819_Error(
	En := TRUE,
	iTerminal_ID := iTerminal_ID,
	bWcState := WcState_WcState,
	uiInfoData_State := InfoData_State,
	pErrorSystem := ErrorSystem,
	bError => bError,
);

IF En THEN
	IF bError=FALSE THEN
		bDi_1:=Channel_1_Input;
		bDi_2:=Channel_2_Input;
		bDi_3:=Channel_3_Input;
		bDi_4:=Channel_4_Input;
		bDi_5:=Channel_5_Input;
		bDi_6:=Channel_6_Input;
		bDi_7:=Channel_7_Input;
		bDi_8:=Channel_8_Input;
		bDi_9:=Channel_9_Input;
		bDi_10:=Channel_10_Input;
		bDi_11:=Channel_11_Input;
		bDi_12:=Channel_12_Input;
		bDi_13:=Channel_13_Input;
		bDi_14:=Channel_14_Input;
		bDi_15:=Channel_15_Input;
		bDi_16:=Channel_16_Input;
	ELSE
		bDi_1:=FALSE;
		bDi_2:=FALSE;
		bDi_3:=FALSE;
		bDi_4:=FALSE;
		bDi_5:=FALSE;
		bDi_6:=FALSE;
		bDi_7:=FALSE;
		bDi_8:=FALSE;
		bDi_9:=FALSE;
		bDi_10:=FALSE;
		bDi_11:=FALSE;
		bDi_12:=FALSE;
		bDi_13:=FALSE;
		bDi_14:=FALSE;
		bDi_15:=FALSE;
		bDi_16:=FALSE;
	END_IF
END_IF

END_FUNCTION_BLOCK

// tc_mca_std_lib/POUs/Hardware/EtherCAT_Terminals/Digital_Inputs/FB_EL1252ASM_v1_00
FUNCTION_BLOCK FB_EL1252ASM_v1_00
VAR_INPUT
	En: BOOL;
END_VAR
VAR_OUTPUT
	EnO: BOOL;
	Di_1: BOOL;
	Di_2: BOOL;
	Di_1_LatchTimePos: ULINT;
	Di_2_LatchTimePos: ULINT;
	Di_1_LatchTimeNeg: ULINT;
	Di_2_LatchTimeNeg: ULINT;
	///Below bits can be used but then they must be enabled in the COE of the card. Nicklas suggested to not use these (since something wss written that you then only were allowed to read the latch time onece (some kkind of auto reset??))	
	///Di_1_LatchNeg:BOOL;
	///	Di_1_LatchPos:BOOL;
	///	Di_2_LatchNeg:BOOL;
	///	Di_2_LatchPos:BOOL;
	Error: BOOL;
END_VAR
VAR
	Channel_1_Input AT %I*: BOOL;
	Channel_2_Input AT %I*: BOOL;
	///Latch_Status1 AT %I*: USINT;
	///	Latch_Status2 AT %I*: USINT;
	Latch_LatchPos1 AT %I*: ULINT;
	Latch_LatchNeg1 AT %I*: ULINT;
	Latch_LatchPos2 AT %I*: ULINT;
	Latch_LatchNeg2 AT %I*: ULINT;
	WcState_WcState AT %I*: BOOL;
	InfoData_State AT %I*: UINT;
END_VAR

EnO:=En;

IF En AND (WcState_WcState OR InfoData_State<>16#8) THEN //InfoData_State==0 => in OP mode
	Error:=TRUE;
ELSE
	Error:=FALSE;
END_IF

IF En THEN
	IF Error=FALSE THEN
		Di_1:=Channel_1_Input;
		Di_2:=Channel_2_Input;
	(*	Di_1_LatchPos:=Latch_Status1.0;
		Di_1_LatchNeg:=Latch_Status1.1;
		Di_2_LatchPos:=Latch_Status2.0;
		Di_2_LatchNeg:=Latch_Status2.1;*)
		Di_1_LatchTimePos:=Latch_LatchPos1;
		Di_2_LatchTimePos:=Latch_LatchPos2;		
		Di_1_LatchTimeNeg:=Latch_LatchNeg1;		
		Di_2_LatchTimeNeg:=Latch_LatchNeg2;
		
	ELSE
		Di_1:=FALSE;
		Di_2:=FALSE;
	END_IF
END_IF

END_FUNCTION_BLOCK

// tc_mca_std_lib/POUs/Hardware/EtherCAT_Terminals/Digital_Outputs/EL2014
FUNCTION_BLOCK EL2014
VAR_INPUT
	En: BOOL;
	iTerminal_ID : INT; 
	bDo_1: BOOL;
	bDo_2: BOOL;
	bDo_3: BOOL;
	bDo_4: BOOL;
	ErrorSystem : POINTER TO ST_ErrorSystem;
END_VAR

VAR_OUTPUT
	EnO : BOOL;
	bError : BOOL;
END_VAR

VAR
	Channel_1_Output AT %Q*: BOOL;
	Channel_2_Output AT %Q*: BOOL;
	Channel_3_Output AT %Q*: BOOL;
	Channel_4_Output AT %Q*: BOOL;
	WcState_WcState AT %I*: BOOL;
	InfoData_State AT %I*: UINT;
	
	//FB-s
	EL2014_Error : FB_TerminalError;
END_VAR

(*
* TODO:
* Channel diagnostic variables and device diag variables
*)

EnO:=En;

EL2014_Error(
	En := TRUE,
	iTerminal_ID := iTerminal_ID,
	bWcState := WcState_WcState,
	uiInfoData_State := InfoData_State,
	pErrorSystem := ErrorSystem,
	bError => bError,
);

IF En THEN
	IF bError=FALSE THEN
		Channel_1_Output:=bDo_1;
		Channel_2_Output:=bDo_2;
		Channel_3_Output:=bDo_3;
		Channel_4_Output:=bDo_4;
	ELSE
		Channel_1_Output:=FALSE;
		Channel_2_Output:=FALSE;
		Channel_3_Output:=FALSE;
		Channel_4_Output:=FALSE;
	END_IF
END_IF

END_FUNCTION_BLOCK

// tc_mca_std_lib/POUs/Hardware/EtherCAT_Terminals/Digital_Outputs/EL2252
///EL2252 | XFC, 2-channel digital output terminal with time stamp, tri-state
FUNCTION_BLOCK EL2252
VAR_INPUT
	En: BOOL;
	iTerminal_ID : INT; 
	bDo_1: BOOL;
	bDo_2: BOOL;
ErrorSystem : POINTER TO ST_ErrorSystem;
END_VAR

VAR_OUTPUT
	EnO : BOOL;
	bError : BOOL;
END_VAR

VAR
	Channel_1_Output AT %Q*: BOOL;
	Channel_2_Output AT %Q*: BOOL;
	WcState_WcState AT %I*: BOOL;
	InfoData_State AT %I*: UINT;
	
	//FB-s
	EL2252_Error : FB_TerminalError;
END_VAR

(*
* TODO:
* Add the DC sync variables
*)

EL2252_Error(
	En := TRUE,
	iTerminal_ID := iTerminal_ID,
	bWcState := WcState_WcState,
	uiInfoData_State := InfoData_State,
	pErrorSystem := ErrorSystem,
	bError => bError,
);

IF En THEN
	IF bError=FALSE THEN
		Channel_1_Output:=bDo_1;
		Channel_2_Output:=bDo_2;
	ELSE
		Channel_1_Output:=FALSE;
		Channel_2_Output:=FALSE;
	END_IF
END_IF

END_FUNCTION_BLOCK

// tc_mca_std_lib/POUs/Hardware/EtherCAT_Terminals/Digital_Outputs/EL2808
FUNCTION_BLOCK EL2808

VAR_INPUT
	En: BOOL;
	iTerminal_ID : INT; 
	bDo_1: BOOL;
	bDo_2: BOOL;
	bDo_3: BOOL;
	bDo_4: BOOL;
	bDo_5: BOOL;
	bDo_6: BOOL;
	bDo_7: BOOL;
	bDo_8: BOOL;
	ErrorSystem : POINTER TO ST_ErrorSystem;
END_VAR

VAR_OUTPUT
	EnO : BOOL;
	bError : BOOL;
END_VAR

VAR
	Channel_1_Output AT %Q*: BOOL;
	Channel_2_Output AT %Q*: BOOL;
	Channel_3_Output AT %Q*: BOOL;
	Channel_4_Output AT %Q*: BOOL;
	Channel_5_Output AT %Q*: BOOL;
	Channel_6_Output AT %Q*: BOOL;
	Channel_7_Output AT %Q*: BOOL;
	Channel_8_Output AT %Q*: BOOL;
	WcState_WcState AT %I*: BOOL;
	InfoData_State AT %I*: UINT;
	
	//FB-s
	EL2808_Error : FB_TerminalError;
END_VAR

EnO:=En;

EL2808_Error(
	En := TRUE,
	iTerminal_ID := iTerminal_ID,
	bWcState := WcState_WcState,
	uiInfoData_State := InfoData_State,
	pErrorSystem := ErrorSystem,
	bError => bError,
);

IF En THEN
	IF bError=FALSE THEN
		Channel_1_Output:=bDo_1;
		Channel_2_Output:=bDo_2;
		Channel_3_Output:=bDo_3;
		Channel_4_Output:=bDo_4;
		Channel_5_Output:=bDo_5;
		Channel_6_Output:=bDo_6;
		Channel_7_Output:=bDo_7;
		Channel_8_Output:=bDo_8;
	ELSE
		Channel_1_Output:=FALSE;
		Channel_2_Output:=FALSE;
		Channel_3_Output:=FALSE;
		Channel_4_Output:=FALSE;
		Channel_5_Output:=FALSE;
		Channel_6_Output:=FALSE;
		Channel_7_Output:=FALSE;
		Channel_8_Output:=FALSE;
	END_IF
END_IF

END_FUNCTION_BLOCK

// tc_mca_std_lib/POUs/Hardware/EtherCAT_Terminals/Digital_Outputs/EL2819
FUNCTION_BLOCK EL2819
VAR_INPUT
	En: BOOL;
	iTerminal_ID : INT; 
	bDo_1: BOOL;
	bDo_2: BOOL;
	bDo_3: BOOL;
	bDo_4: BOOL;
	bDo_5: BOOL;
	bDo_6: BOOL;
	bDo_7: BOOL;
	bDo_8: BOOL;
	bDo_9: BOOL;
	bDo_10: BOOL;
	bDo_11: BOOL;
	bDo_12: BOOL;
	bDo_13: BOOL;
	bDo_14: BOOL;
	bDo_15: BOOL;
	bDo_16: BOOL;
	ErrorSystem : POINTER TO ST_ErrorSystem;
END_VAR

VAR_OUTPUT
	EnO : BOOL;
	bError : BOOL;
END_VAR

VAR
	Channel_1_Output AT %Q*: BOOL;
	Channel_2_Output AT %Q*: BOOL;
	Channel_3_Output AT %Q*: BOOL;
	Channel_4_Output AT %Q*: BOOL;
	Channel_5_Output AT %Q*: BOOL;
	Channel_6_Output AT %Q*: BOOL;
	Channel_7_Output AT %Q*: BOOL;
	Channel_8_Output AT %Q*: BOOL;
	Channel_9_Output AT %Q*: BOOL;
	Channel_10_Output AT %Q*: BOOL;
	Channel_11_Output AT %Q*: BOOL;
	Channel_12_Output AT %Q*: BOOL;
	Channel_13_Output AT %Q*: BOOL;
	Channel_14_Output AT %Q*: BOOL;
	Channel_15_Output AT %Q*: BOOL;
	Channel_16_Output AT %Q*: BOOL;
	
	WcState_WcState AT %I*: BOOL;
	InfoData_State AT %I*: UINT;
	
	//FB-s
	EL2819_Error : FB_TerminalError;
END_VAR

(*
* TODO:
* Channel diagnostic variables and device diag variables
*)

EnO:=En;

EL2819_Error(
	En := TRUE,
	iTerminal_ID := iTerminal_ID,
	bWcState := WcState_WcState,
	uiInfoData_State := InfoData_State,
	pErrorSystem := ErrorSystem,
	bError => bError,
);

IF En THEN
	IF bError=FALSE THEN
		Channel_1_Output:=bDo_1;
		Channel_2_Output:=bDo_2;
		Channel_3_Output:=bDo_3;
		Channel_4_Output:=bDo_4;
		Channel_5_Output:=bDo_5;
		Channel_6_Output:=bDo_6;
		Channel_7_Output:=bDo_7;
		Channel_8_Output:=bDo_8;
		Channel_9_Output:=bDo_9;
		Channel_10_Output:=bDo_10;
		Channel_11_Output:=bDo_11;
		Channel_12_Output:=bDo_12;
		Channel_13_Output:=bDo_13;
		Channel_14_Output:=bDo_14;
		Channel_15_Output:=bDo_15;
		Channel_16_Output:=bDo_16;
	ELSE
		Channel_1_Output:=FALSE;
		Channel_2_Output:=FALSE;
		Channel_3_Output:=FALSE;
		Channel_4_Output:=FALSE;
		Channel_5_Output:=FALSE;
		Channel_6_Output:=FALSE;
		Channel_7_Output:=FALSE;
		Channel_8_Output:=FALSE;
		Channel_9_Output:=FALSE;
		Channel_10_Output:=FALSE;
		Channel_11_Output:=FALSE;
		Channel_12_Output:=FALSE;
		Channel_13_Output:=FALSE;
		Channel_14_Output:=FALSE;
		Channel_15_Output:=FALSE;
		Channel_16_Output:=FALSE;
	END_IF
END_IF

END_FUNCTION_BLOCK

// tc_mca_std_lib/POUs/Hardware/EtherCAT_Terminals/Measuring_Terminals/EL5002
//EL5002 | 2-chennel SSI absolute encoder terminal
FUNCTION_BLOCK EL5002

VAR_INPUT
	En: BOOL;
	iTerminal_ID : INT;
	ErrorSystem : POINTER TO ST_ErrorSystem;
END_VAR

VAR_OUTPUT
	EnO: BOOL;
	Ch1_Counter_Value : UDINT;
	Ch2_Counter_Value : UDINT;
	bError: BOOL;
END_VAR

VAR
	udi_Ch1_Cnt_Value AT %I* : UDINT;
	udi_Ch2_Cnt_Value AT %I* : UDINT;
	WcState_WcState AT %I*: BOOL;
	InfoData_State AT %I*: UINT;
	
	//FB-s
	EL5002_Error : FB_TerminalError;
END_VAR

(*
* TODO:
* Channel Status words
*)

EnO:=En;

//Error FB instance
EL5002_Error(
	En := TRUE,
	iTerminal_ID := iTerminal_ID,
	bWcState := WcState_WcState,
	uiInfoData_State := InfoData_State,
	pErrorSystem := ErrorSystem,
	bError => bError,
);

IF EN THEN
	IF NOT bError THEN
		Ch1_Counter_Value := udi_Ch1_Cnt_Value;
		Ch2_Counter_Value := udi_Ch2_Cnt_Value;
	ELSE
		Ch1_Counter_Value := 0;
		Ch2_Counter_Value := 0;
	END_IF
END_IF

END_FUNCTION_BLOCK

// tc_mca_std_lib/POUs/Hardware/EtherCAT_Terminals/Measuring_Terminals/EL5021
//EL5021 | 1-channel Sin/Cos encoder
FUNCTION_BLOCK EL5021

VAR_INPUT
	En: BOOL;
	iTerminal_ID : INT;
	ErrorSystem : POINTER TO ST_ErrorSystem;
END_VAR

VAR_OUTPUT
	EnO: BOOL;
	Counter_Value : UDINT;
	Latch_Value : UDINT;
	bError: BOOL;
END_VAR

VAR
	udiCounter_Value AT %I* : UDINT;
	udiLatch_Value AT %I* : UDINT;
	WcState_WcState AT %I*: BOOL;
	InfoData_State AT %I*: UINT;
	
	//FB-s
	EL5021_Error : FB_TerminalError;
END_VAR

(*
* TODO:
* Channel Status words, control words
*)

EnO:=En;

//Error FB instance
EL5021_Error(
	En := TRUE,
	iTerminal_ID := iTerminal_ID,
	bWcState := WcState_WcState,
	uiInfoData_State := InfoData_State,
	pErrorSystem := ErrorSystem,
	bError => bError,
);

IF EN THEN
	IF NOT bError THEN
		Counter_Value := udiCounter_Value;
		Latch_Value := udiLatch_Value;
	ELSE
		Counter_Value := 0;
		Latch_Value := 0;
	END_IF
END_IF

END_FUNCTION_BLOCK

// tc_mca_std_lib/POUs/Hardware/EtherCAT_Terminals/Measuring_Terminals/EL5042
//EL5042 | 2-channel BiSS-C absolute encoder terminal
FUNCTION_BLOCK EL5042

VAR_INPUT
	En: BOOL;
	iTerminal_ID : INT;
	ErrorSystem : POINTER TO ST_ErrorSystem;
END_VAR

VAR_OUTPUT
	EnO: BOOL;
	Ch1_Position : ULINT;
	Ch2_Position : ULINT;
	bError: BOOL;
END_VAR

VAR
	FB_Inputs_ch1_Position AT %I* : ULINT;
	FB_Inputs_ch2_Position AT %I* : ULINT;
	WcState_WcState AT %I*: BOOL;
	InfoData_State AT %I*: UINT;
	
	//FB-s
	EL5042_Error : FB_TerminalError;
END_VAR

(*
* TODO:
* Channel Status words
*)

EnO:=En;

//Error FB instance
EL5042_Error(
	En := TRUE,
	iTerminal_ID := iTerminal_ID,
	bWcState := WcState_WcState,
	uiInfoData_State := InfoData_State,
	pErrorSystem := ErrorSystem,
	bError => bError,
);

IF EN THEN
	IF NOT bError THEN
		Ch1_Position := FB_Inputs_ch1_Position;
		Ch2_Position := FB_Inputs_ch2_Position;
	ELSE
		Ch1_Position := 0;
		Ch2_Position := 0;
	END_IF
END_IF

END_FUNCTION_BLOCK

// tc_mca_std_lib/POUs/Hardware/EtherCAT_Terminals/Measuring_Terminals/EL5101
// EL5101 | 1-channel incremental encoder terminal, 5V, RS422
FUNCTION_BLOCK EL5101

VAR_INPUT
	En: BOOL;
	iTerminal_ID : INT;
	ErrorSystem : POINTER TO ST_ErrorSystem;
END_VAR

VAR_OUTPUT
	EnO: BOOL;
	Counter_Value : UINT;
	Latch_Value : UINT;
	bError: BOOL;
END_VAR

VAR
	uiCounter_Value AT %I* : UINT;
	uiLatch_Value AT %I* : UINT;
	WcState_WcState AT %I*: BOOL;
	InfoData_State AT %I*: UINT;
	
	//FB-s
	EL5101_Error : FB_TerminalError;
END_VAR

(*
* TODO:
* Channel Status word, control words
*)

EnO:=En;

//Error FB instance
EL5101_Error(
	En := TRUE,
	iTerminal_ID := iTerminal_ID,
	bWcState := WcState_WcState,
	uiInfoData_State := InfoData_State,
	pErrorSystem := ErrorSystem,
	bError => bError,
);

IF EN THEN
	IF NOT bError THEN
		Counter_Value := uiCounter_Value;
		Latch_Value := uiLatch_Value;
	ELSE
		Counter_Value := 0;
		Latch_Value := 0;
	END_IF
END_IF

END_FUNCTION_BLOCK

// tc_mca_std_lib/POUs/Hardware/EtherCAT_Terminals/Motion/EL7211_v1_00
///EL7211 | Servo motor termional 5 A
FUNCTION_BLOCK EL7211_v1_00
VAR_INPUT
	En: BOOL;
END_VAR
VAR_OUTPUT
	EnO: BOOL;

	bError: BOOL;
END_VAR
VAR
	WcState_WcState AT %I*: BOOL;
	InfoData_State AT %I*: UINT;
END_VAR

EnO:=En;

IF En AND (WcState_WcState OR InfoData_State<>16#8) THEN
	bError:=TRUE;
ELSE
	bError:=FALSE;
END_IF

END_FUNCTION_BLOCK

// tc_mca_std_lib/POUs/Hardware/EtherCAT_Terminals/Motion/EL9576_v1_00
///EL9576 | Brake terminal (vap and resistor)
FUNCTION_BLOCK EL9576_v1_00
VAR_INPUT
	En: BOOL;
END_VAR
VAR_OUTPUT
	EnO: BOOL;
	bError: BOOL;	
	OverTemperature: BOOL;
	I2TError : BOOL;
	I2TWarning : BOOL;
	OverVoltage  : BOOL;
	UnderVoltage : BOOL;
	ChopperOn : BOOL;
	DCLinkVoltage : LREAL;
	DutyCycle  : LREAL;
	ResistorCurrent : LREAL;
	
END_VAR
VAR
	BCTOverTemperature AT %I*: BOOL;
	BCTI2TError AT %I*: BOOL;
	BCTI2TWarning AT %I*: BOOL;
	BCTOverVoltage  AT %I*: BOOL;
	BCTUnderVoltage  AT %I*: BOOL;
	BCTChopperOn  AT %I*: BOOL;
	BCTDCLinkVoltage AT %I*: UDINT;
	BCTDutyCycle  AT %I*: USINT;
	BCTResistorCurrent AT %I*: UDINT;
	WcState_WcState AT %I*: BOOL;
	InfoData_State AT %I*: UINT;
	
END_VAR

EnO:=En;

IF En AND (WcState_WcState OR InfoData_State<>16#8 OR BCTI2TError OR BCTI2TWarning OR BCTOverTemperature OR BCTOverVoltage OR BCTUnderVoltage) THEN
	bError:=TRUE;
ELSE
	bError:=FALSE;
END_IF

OverTemperature:=BCTOverTemperature;
I2TError:=BCTI2TError;
I2TWarning:=BCTI2TWarning;
OverVoltage:=BCTOverVoltage;
UnderVoltage:=bctUnderVoltage;
ChopperOn:=bctChopperOn;
DCLinkVoltage:=UDINT_TO_LREAL(bctDCLinkVoltage);
DutyCycle:=USINT_TO_LREAL(BCTDutyCycle);
ResistorCurrent:=UDINT_TO_LREAL(BCTResistorCurrent);

END_FUNCTION_BLOCK

// tc_mca_std_lib/POUs/Hardware/EtherCAT_Terminals/System/EL9410
//EL9410 | E-Bus power supplier and refresher, diagnostics
FUNCTION_BLOCK EL9410

VAR_INPUT
	En: BOOL;
	iTerminal_ID : INT;
	ErrorSystem : POINTER TO ST_ErrorSystem;
END_VAR

VAR_OUTPUT
	EnO: BOOL;
	bError: BOOL;
END_VAR

VAR
	bStatus_Us_UV AT %I* : BOOL;
	bStatus_Up_UV AT %I* : BOOL;
	WcState_WcState AT %I*: BOOL;
	InfoData_State AT %I*: UINT;
	
	//FB-s
	EL9410_Error : FB_TerminalError;
END_VAR

(*
* TODO:
* Status bits
*)

EnO:=En;

//Error FB instance
EL9410_Error(
	En := TRUE,
	iTerminal_ID := iTerminal_ID,
	bWcState := WcState_WcState,
	uiInfoData_State := InfoData_State,
	pErrorSystem := ErrorSystem,
	bError => bError,
);

END_FUNCTION_BLOCK

// tc_mca_std_lib/POUs/Hardware/EtherCAT_Terminals/System/EL9505
//EL9505 | Power supply terminal 5V
FUNCTION_BLOCK EL9505

VAR_INPUT
	En: BOOL;
	iTerminal_ID : INT;
	ErrorSystem : POINTER TO ST_ErrorSystem;
END_VAR

VAR_OUTPUT
	EnO: BOOL;
	bError: BOOL;
END_VAR

VAR
	bStatus_Uo_Power_OK AT %I* : BOOL;
	bStatus_Uo_Overload AT %I* : BOOL;
	WcState_WcState AT %I*: BOOL;
	InfoData_State AT %I*: UINT;
	
	//FB-s
	EL9505_Error : FB_TerminalError;
END_VAR

(*
* TODO:
* Status bits
*)
EnO:=En;

//Error FB instance
EL9505_Error(
	En := TRUE,
	iTerminal_ID := iTerminal_ID,
	bWcState := WcState_WcState,
	uiInfoData_State := InfoData_State,
	pErrorSystem := ErrorSystem,
	bError => bError,
);

END_FUNCTION_BLOCK

// tc_mca_std_lib/POUs/Hardware/Other/EK1200
FUNCTION_BLOCK EK1200
VAR_INPUT
	En: BOOL;
END_VAR
VAR_OUTPUT
	EnO: BOOL;
END_VAR

EnO:=En;

END_FUNCTION_BLOCK

// tc_mca_std_lib/POUs/Motion/FB_NcAxis
///#########################################################
///Function block to communicate between Nc and Plc.
///
///	Library:		
///	Tc2_MC2.lib
///
///	Global Variables:
///	
///	Data types:
///	
///	External functions:
///
///###########################################################
FUNCTION_BLOCK FB_NcAxis
VAR
	sVersion: STRING:='1.0.0';
END_VAR
VAR_INPUT
	En: BOOL;
END_VAR
VAR_OUTPUT
	EnO: BOOL;
	bError: BOOL;
	Status: ST_AxisStatus;
END_VAR
VAR
	Axis: AXIS_REF;
	InfoData_State AT %I*: UINT;
END_VAR

EnO:=En;

IF En AND InfoData_State<>16#8 THEN
	bError:=TRUE;
ELSE
	bError:=FALSE;
END_IF

IF En THEN
	Axis.ReadStatus();
	Status:=Axis.Status;
END_IF

END_FUNCTION_BLOCK

// UnitTests/BasicTests
PROGRAM BasicTests
VAR
    Motor: DUT_MotionStage;
    fbMotion: FB_MotionStageSim;
    fbRequest: FB_MotionRequest;

    bError: BOOL;
    errState: MC_AxisStates;
END_VAR

fbRequest(stMotionStage := Motor);
fbMotion(stMotionStage := Motor);

CASE Motor.Axis.Status.MotionState OF
   MC_AXISSTATE_ERRORSTOP,
   MC_AXISSTATE_STOPPING,
   MC_AXISSTATE_HOMING,
   MC_AXISSTATE_DISCRETEMOTION,
   MC_AXISSTATE_CONTINOUSMOTION,
   MC_AXISSTATE_SYNCHRONIZEDMOTION:
        IF NOT Motor.bBrakeRelease THEN
            bError := TRUE;
            errState := Motor.Axis.Status.MotionState;
        END_IF
END_CASE

END_PROGRAM

// UnitTests/Interactive
PROGRAM Interactive
VAR
    bInit: BOOL := FALSE;

    M1: DUT_MotionStage;
    fbMotionStageSim: FB_MotionStageSim;
    nCounter: UINT;

    stOut: DUT_PositionState;
    fbGoOut: FB_PositionStateMove;
    bOut: BOOL;
    bGoOut: BOOL;
    stIn: DUT_PositionState;
    fbGoIn: FB_PositionStateMove;
    bIn: BOOL;
    bGoIn: BOOL;
    stUnsafe: DUT_PositionState;
    fbGoBad: FB_PositionStateMove;
    bHCF: BOOL;
    bGoHCF: BOOL;

    {attribute 'pytmc' := '
        pv: TST:STATE
        io: io
    '}
    fbEpicsInOut: FB_EpicsInOut;

    fbStateManager: FB_PositionStateManager;
    setState: INT;
    arrStates: ARRAY [1..15] OF DUT_PositionState;
END_VAR

BasicTests();

fbMotionStageSim(stMotionStage:=M1);
nCounter := nCounter + 1;

IF NOT bInit THEN
    bInit := TRUE;

    stOut.sName := 'Out';
    stOut.fPosition := 100;
    stOut.fDelta := 20;
    stOut.fVelocity := 10;
    stOut.bValid := TRUE;
    stOut.bMoveOk := TRUE;

    stIn.sName := 'In';
    stIn.fPosition := 0;
    stIn.fDelta := 0.1;
    stIn.fVelocity := 5;
    stIn.bValid := TRUE;
    stIn.bMoveOk := TRUE;

    stUnsafe.sName := 'HCF';
    stUnsafe.fPosition := -999;
    stUnsafe.fDelta := 6;
    stUnsafe.fVelocity := 42;
    stUnsafe.bValid := TRUE;
    stUnsafe.bMoveOk := FALSE;

    fbEpicsInOut.bEnable := TRUE;
    fbStateManager.bEnable := TRUE;
END_IF

fbGoOut(
    bExecute:=bGoOut,
    stMotionStage:=M1,
    stPositionState:=stOut,
    bAtState=>bOut);
fbGoIn(
    bExecute:=bGoIn,
    stMotionStage:=M1,
    stPositionState:=stIn,
    bAtState=>bIn);
fbGoBad(
    bExecute:=bGoHCF,
    stMotionStage:=M1,
    stPositionState:=stUnsafe,
    bAtState=>bHCF);

arrStates[1] := stOut;
arrStates[2] := stIn;
arrStates[3] := stUnsafe;

fbEpicsInOut(
    stMotionStage := M1,
    stOut := stOut,
    stIn := stIn);

fbStateManager(
    stMotionStage := M1,
    arrStates := arrStates,
    setState := setState);

END_PROGRAM
